(* CODESYS project Defaults.gvl.xml

Project tree, tasks and I/O mapping:
  global variables Defaults
*)

// Defaults
{attribute 'qualified_only'}
VAR_GLOBAL
	
END_VAR
